Fanuc KAREL source: compact_preamble.KL

PROGRAM KT00602
%NOLOCKGROUP
VAR
I1:INTEGER;I2:INTEGER;OUT:REAL
BEGIN
I1=2
I2=3
I1=2
I2=3
OUT=(I1)
END KT00602
